TEXTLIST nNCEventTableHeader
  0 = 'Eksen' | English: 'Axis ID' | Turkish: 'Eksen'
  1 = 'Hata Kodu' | English: 'Error ID' | Turkish: 'Hata Kodu'
  2 = 'Mesaj' | English: 'Message' | Turkish: 'Mesaj'
  3 = 'Zaman' | English: 'Event Time' | Turkish: 'Zaman'
  4 = 'Onay' | English: 'Ack Time' | Turkish: 'Onay'
   = ''
END_TEXTLIST

(* stored: Version 1.1.0.1, ProductVersion 3.1.4024.6
   TextList nNCEventTableHeader: Id {6e04746a-3378-456e-8e3b-38ce1ea78d64} *)
